Universal Robots PolyScope program: RC_E3_PLACE_330.urp

Program RC_E3_PLACE_330 (createdIn=3.0.0 lastSavedIn=3.0.0 directory=/programs installation=default)
Robot Program (runOnlyOnce=true motionType=MoveJ speed=1.047198 acceleration=1.396263 useActiveTCP=false)
  'Program generated by RoboDK v4.1.0 for UR3e_HORNO on 27/07/2022 12:03:32'
  'Using nominal kinematics.'
  'Using Ref. Frame Horno: p[0.203000, 0.332000, 0.148000, 0.000000, 0.000000, 0.000000]'
  'Using TCP 0208-0001-0001-307-000-3 Horno: p[0.000000, 0.000000, 0.038000, 0.000000, 0.000000, 0.000000]'
  Script: set_tcp(p[0.000000, 0.000000, 0.038000, 0.000000, 0.000000, 0.000000])
  Script: movej([1.826764, -1.419904, -1.065151, -2.231914, 1.547896, 0.233255],0.60000,0.12500,0,0.0000)
  Script: movej([1.925098, -2.178520, -0.657466, -1.883210, 1.548456, 0.331613],0.60000,0.12500,0,0.0000)
  MoveL speed 100 mm/s, acceleration 120 mm/s^2 (useActiveTCP=true)
    Waypoint Waypoint_1: TCP in base x=190.053 y=818.549 z=350.19 mm, rx=3.138 ry=-0.0211 rz=0.0107 rad; joints [107.23, -134.54, -43.51, -92.26, 89.69, 18] deg; flange x=189.796 y=818.684 z=388.188 mm, rx=3.138 ry=-0.0211 rz=0.0107 rad
  'Detach from 0208-0001-0001-307-000-4 Horno'
  MoveL speed 500 mm/s, acceleration 900 mm/s^2 (useActiveTCP=true)
    Waypoint Waypoint_2: TCP in base x=180.546 y=778.813 z=433.343 mm, rx=-3.1401 ry=-0.0357 rz=-0.0366 rad; joints [110.3, -124.82, -37.67, -107.9, 88.72, 19] deg; flange x=179.66 y=778.761 z=471.332 mm, rx=-3.1401 ry=-0.0357 rz=-0.0366 rad
  Script: movej([1.826764, -1.419904, -1.065151, -2.231914, 1.547896, 0.233255],0.90000,0.50000,0,0.0000)
